(* Schneider Machine Expert - Basic project Pompa Otomatis dan Manual Fungsion Blok, file version 1.7.0.0 *)
(* ProjectInformations: Name=New project *)

HARDWARE
  Cpu 0: TM221M16R/G
  EthernetConfiguration: NetworkName=M221, IpAllocationMode=FixedAddress, IpAddress=0.0.0.0, SubnetMask=0.0.0.0
  SerialLineConfiguration: Baud=Baud19200, Parity=ParityEven, DataBits=DataBits8, StopBits=StopBits1, PhysicalMedium=PhysicalMediumRs485, TransmissionMode=TransmissionModeModbusRtu, SlaveId=1, Addressing=SlaveAddressing
  MastTask: UsePeriodScanMode=false, PeriodScan=100
  FastTask: Period=255
  CpuBehavior: StartingMode=StartAsPreviousState, AutoSaveRamOnEeprom=true, WatchdogPeriod=250

SYMBOLS  (address, symbol, comment, settings)
  %TM0        [Preset=5, Base=OneSecond]
  %TM1        [Preset=5, Base=OneSecond]
  %TM2        [Preset=5, Base=OneSecond, IsRetentive=true]
  %TM3        [Preset=5, Base=OneSecond, IsRetentive=true]
  %TM4        [Preset=60, Base=OneSecond, IsRetentive=true]
  %TM5        [Preset=60, Base=OneSecond, IsRetentive=true]
  %I0.0       "Auto"
  %I0.1       "MAN"
  %I0.2       "POM A"
  %I0.3       "POM B"
  %Q0.0       "POMPA A"
  %Q0.1       "POMPA B"

POU New POU
  (* SectionNumber=1 *)

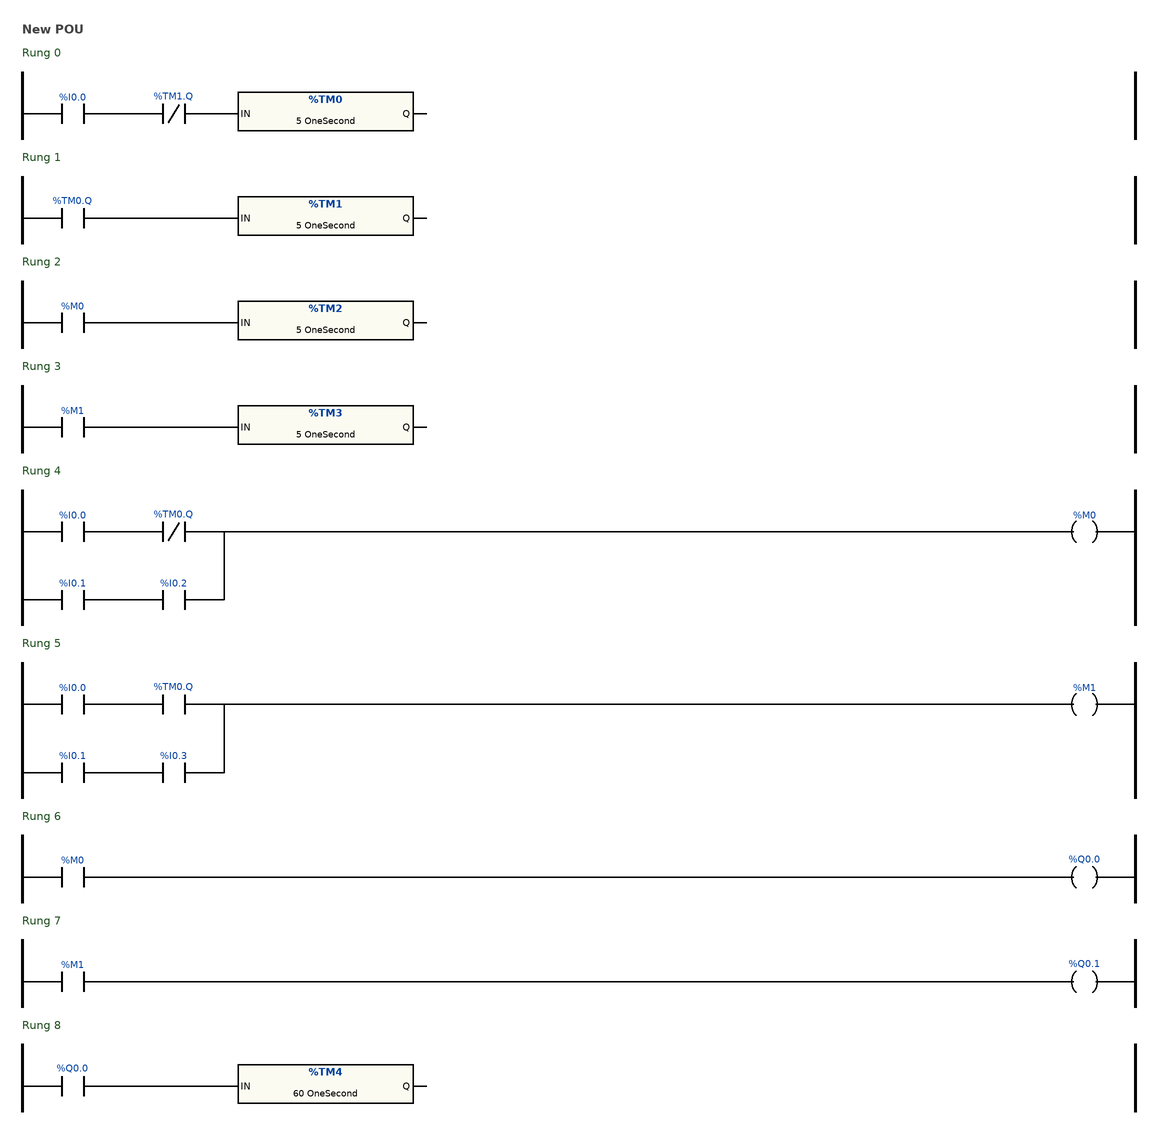

// Rung 0
  BLK %TM0
  LD %I0.0
  ANDN %TM1.Q
  IN
  END_BLK
  // as ST:
  //   %TM0(IN := %I0.0 AND NOT %TM1.Q);

// Rung 1
  BLK %TM1
  LD %TM0.Q
  IN
  END_BLK
  // as ST:
  //   %TM1(IN := %TM0.Q);

// Rung 2
  BLK %TM2
  LD %M0
  IN
  END_BLK
  // as ST:
  //   %TM2(IN := %M0);

// Rung 3
  BLK %TM3
  LD %M1
  IN
  END_BLK
  // as ST:
  //   %TM3(IN := %M1);

// Rung 4
  LD %I0.0
  ANDN %TM0.Q
  OR( %I0.1
  AND %I0.2
  )
  ST %M0
  // as ST:
  //   %M0 := %I0.0 AND NOT %TM0.Q OR %I0.1 AND %I0.2;

// Rung 5
  LD %I0.0
  AND %TM0.Q
  OR( %I0.1
  AND %I0.3
  )
  ST %M1
  // as ST:
  //   %M1 := %I0.0 AND %TM0.Q OR %I0.1 AND %I0.3;

// Rung 6
  LD %M0
  ST %Q0.0
  // as ST:
  //   %Q0.0 := %M0;

// Rung 7
  LD %M1
  ST %Q0.1
  // as ST:
  //   %Q0.1 := %M1;

// Rung 8
  BLK %TM4
  LD %Q0.0
  IN
  END_BLK
  // as ST:
  //   %TM4(IN := %Q0.0);

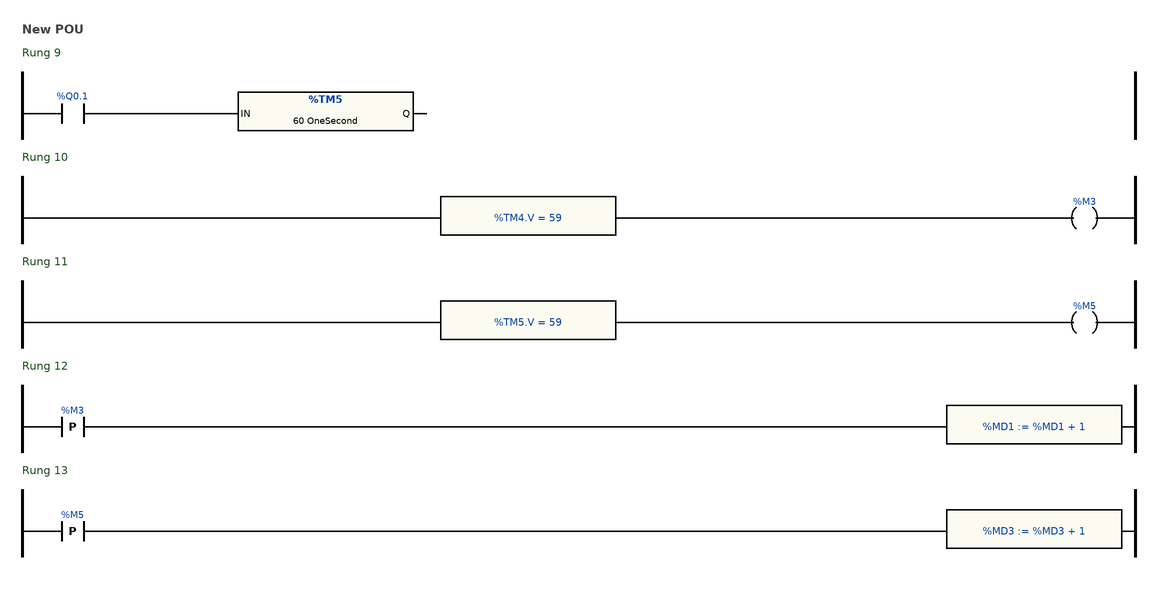

// Rung 9
  BLK %TM5
  LD %Q0.1
  IN
  END_BLK
  // as ST:
  //   %TM5(IN := %Q0.1);

// Rung 10
  LD [ %TM4.V = 59 ]
  ST %M3
  // as ST:
  //   %M3 := %TM4.V = 59;

// Rung 11
  LD [ %TM5.V = 59 ]
  ST %M5
  // as ST:
  //   %M5 := %TM5.V = 59;

// Rung 12
  LDR %M3
  [ %MD1 := %MD1 + 1 ]
  // as ST:
  //   IF RISING(%M3) THEN %MD1 := %MD1 + 1; END_IF;

// Rung 13
  LDR %M5
  [ %MD3 := %MD3 + 1 ]
  // as ST:
  //   IF RISING(%M5) THEN %MD3 := %MD3 + 1; END_IF;
